FUNCTION_BLOCK CM_DO_3state_CALL
VAR_INPUT
END_VAR
VAR_OUTPUT
END_VAR
VAR
	
END_VAR

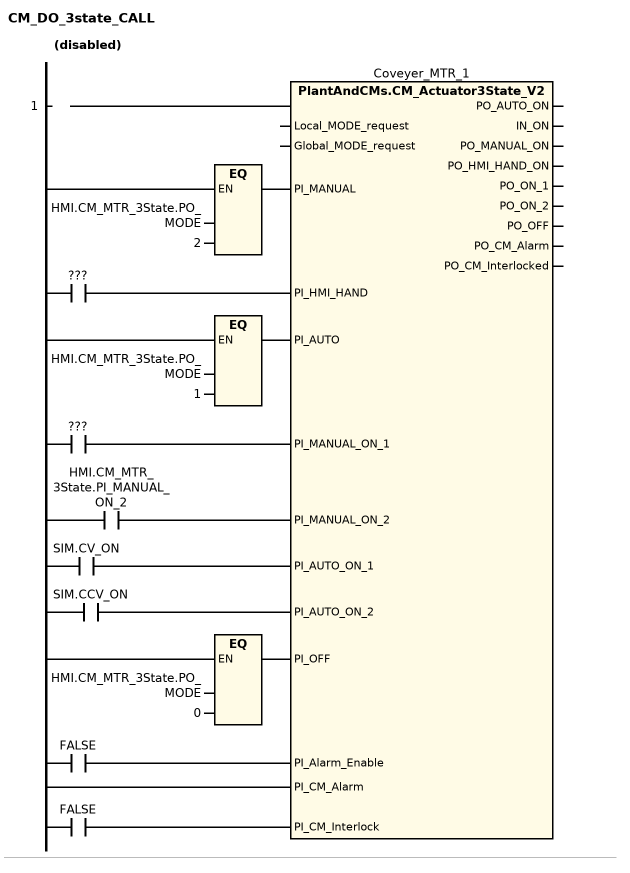
// NETWORK 1 (disabled)
// Coveyer_MTR_1(
//     PI_MANUAL := HMI.CM_MTR_3State.PO_MODE = 2,
//     PI_AUTO := HMI.CM_MTR_3State.PO_MODE = 1,
//     PI_MANUAL_ON_2 := HMI.CM_MTR_3State.PI_MANUAL_ON_2,
//     PI_AUTO_ON_1 := SIM.CV_ON,
//     PI_AUTO_ON_2 := SIM.CCV_ON,
//     PI_OFF := HMI.CM_MTR_3State.PO_MODE = 0,
//     PI_Alarm_Enable := FALSE,
//     PI_CM_Alarm := TRUE,
//     PI_CM_Interlock := FALSE); // PlantAndCMs.CM_Actuator3State_V2

END_FUNCTION_BLOCK

(* stored: Version 1.1.0.1, ProductVersion 3.1.4024.13
   POU CM_DO_3state_CALL: Id {b0438b32-cd77-4d2f-8999-4734990b3513}, SpecialFunc None *)
